TYPE ST_Zaptec_Input_Installation :
STRUCT
	rAvailableCurrentInstallation		: REAL;													//Available Current for Installation
	sInstallationID						: STRING(50);											//Installation ID
END_STRUCT
END_TYPE

(* stored: Version 1.1.0.1, ProductVersion 3.1.4024.9
   DUT ST_Zaptec_Input_Installation: Id {4b176467-ea0e-49bb-927b-9eaf410f56ee} *)
